(* PLC project tri_chain, Dassault Systèmes ControlBuild 2024x *)
(* stored: creationDateTime 2023-10-05T15:45:14-01:00 *)

CONFIGURATION tri_chain
  VAR_GLOBAL
    simuperiod : REAL := 50000.0;
    taskname : STRING(50) := 'tri_chain.exe';
    allowpreconditions : BOOL := true;
    allowpostconditions : BOOL := true;
    op_trichain/creation1/status_act_prod : DINT := 0;
    op_trichain/creation1/m11 : REAL := 1502.68;
    op_trichain/creation1/m12 : REAL := 0.0;
    op_trichain/creation1/m13 : REAL := -2.44921e-14;
    op_trichain/creation1/m14 : REAL := 5480.36;
    op_trichain/creation1/m21 : REAL := 0.0;
    op_trichain/creation1/m22 : REAL := 2997.32;
    op_trichain/creation1/m23 : REAL := 0.0;
    op_trichain/creation1/m24 : REAL := 27006.2;
    op_trichain/creation1/m31 : REAL := 3.68038e-13;
    op_trichain/creation1/m32 : REAL := 0.0;
    op_trichain/creation1/m33 : REAL := 100.0;
    op_trichain/creation1/m34 : REAL := 1.0;
    op_trichain/creation1/m41 : REAL := 0.0;
    op_trichain/creation1/m42 : REAL := 0.0;
    op_trichain/creation1/m43 : REAL := 0.0;
    op_trichain/creation1/m44 : REAL := 1.0;
    op_trichain/creation1/px : REAL := 5600.0;
    op_trichain/creation1/py : REAL := 27000.0;
    op_trichain/creation1/pz : REAL := 1.5;
    op_trichain/creation1/dx : REAL := 1500.0;
    op_trichain/creation1/dy : REAL := 3000.0;
    op_trichain/creation1/dz : REAL := 100.0;
    op_trichain/creation1/pulseType : BOOL := true;
    op_trichain/chain1/motor1dir/nominalSpeed : REAL := 500.0;
    op_trichain/chain1/motor1dir/nominalTime : REAL := 0.1;
    op_trichain/chain1/start_sensor/status_act_prod : DINT := 0;
    op_trichain/chain1/start_sensor/m11 : REAL := 498.214;
    op_trichain/chain1/start_sensor/m12 : REAL := 0.0;
    op_trichain/chain1/start_sensor/m13 : REAL := -2.44921e-14;
    op_trichain/chain1/start_sensor/m14 : REAL := 5223.22;
    op_trichain/chain1/start_sensor/m21 : REAL := 0.0;
    op_trichain/chain1/start_sensor/m22 : REAL := 498.214;
    op_trichain/chain1/start_sensor/m23 : REAL := 0.0;
    op_trichain/chain1/start_sensor/m24 : REAL := 26998.2;
    op_trichain/chain1/start_sensor/m31 : REAL := 1.22023e-13;
    op_trichain/chain1/start_sensor/m32 : REAL := 0.0;
    op_trichain/chain1/start_sensor/m33 : REAL := 100.0;
    op_trichain/chain1/start_sensor/m34 : REAL := 1.0;
    op_trichain/chain1/start_sensor/m41 : REAL := 0.0;
    op_trichain/chain1/start_sensor/m42 : REAL := 0.0;
    op_trichain/chain1/start_sensor/m43 : REAL := 0.0;
    op_trichain/chain1/start_sensor/m44 : REAL := 1.0;
    op_trichain/chain1/start_sensor/px : REAL := 4500.0;
    op_trichain/chain1/start_sensor/py : REAL := 27000.0;
    op_trichain/chain1/start_sensor/dx : REAL := 500.0;
    op_trichain/chain1/start_sensor/dy : REAL := 500.0;
    op_trichain/chain1/start_sensor/dz : REAL := 100.0;
    op_trichain/chain1/end_sensor/status_act_prod : DINT := 0;
    op_trichain/chain1/end_sensor/m11 : REAL := 498.214;
    op_trichain/chain1/end_sensor/m12 : REAL := 0.0;
    op_trichain/chain1/end_sensor/m13 : REAL := -2.44921e-14;
    op_trichain/chain1/end_sensor/m14 : REAL := 3334.82;
    op_trichain/chain1/end_sensor/m21 : REAL := 0.0;
    op_trichain/chain1/end_sensor/m22 : REAL := 498.214;
    op_trichain/chain1/end_sensor/m23 : REAL := 0.0;
    op_trichain/chain1/end_sensor/m24 : REAL := 19999.1;
    op_trichain/chain1/end_sensor/m31 : REAL := 1.22023e-13;
    op_trichain/chain1/end_sensor/m32 : REAL := 0.0;
    op_trichain/chain1/end_sensor/m33 : REAL := 100.0;
    op_trichain/chain1/end_sensor/m34 : REAL := 1.05;
    op_trichain/chain1/end_sensor/m41 : REAL := 0.0;
    op_trichain/chain1/end_sensor/m42 : REAL := 0.0;
    op_trichain/chain1/end_sensor/m43 : REAL := 0.0;
    op_trichain/chain1/end_sensor/m44 : REAL := 1.0;
    op_trichain/chain1/end_sensor/px : REAL := 2850.0;
    op_trichain/chain1/end_sensor/py : REAL := 20000.0;
    op_trichain/chain1/end_sensor/dx : REAL := 500.0;
    op_trichain/chain1/end_sensor/dy : REAL := 500.0;
    op_trichain/chain1/end_sensor/dz : REAL := 100.0;
    op_trichain/chain1/chain/status_act_prod : DINT := 0;
    op_trichain/chain1/chain/m11 : REAL := 4001.79;
    op_trichain/chain1/chain/m12 : REAL := 0.0;
    op_trichain/chain1/chain/m13 : REAL := -2.44921e-14;
    op_trichain/chain1/chain/m14 : REAL := 2981.25;
    op_trichain/chain1/chain/m21 : REAL := 0.0;
    op_trichain/chain1/chain/m22 : REAL := 9996.43;
    op_trichain/chain1/chain/m23 : REAL := 0.0;
    op_trichain/chain1/chain/m24 : REAL := 18102.7;
    op_trichain/chain1/chain/m31 : REAL := 9.80123e-13;
    op_trichain/chain1/chain/m32 : REAL := 0.0;
    op_trichain/chain1/chain/m33 : REAL := 100.0;
    op_trichain/chain1/chain/m34 : REAL := 1.0;
    op_trichain/chain1/chain/m41 : REAL := 0.0;
    op_trichain/chain1/chain/m42 : REAL := 0.0;
    op_trichain/chain1/chain/m43 : REAL := 0.0;
    op_trichain/chain1/chain/m44 : REAL := 1.0;
    op_trichain/chain1/chain/px : REAL := 2500.0;
    op_trichain/chain1/chain/py : REAL := 18100.0;
    op_trichain/chain1/chain/pz : REAL := 1.0;
    op_trichain/chain1/chain/dx : REAL := 4000.0;
    op_trichain/chain1/chain/dy : REAL := 10000.0;
    op_trichain/chain1/chain/dz : REAL := 100.0;
    op_trichain/chain2/motor1dir/nominalSpeed : REAL := 500.0;
    op_trichain/chain2/motor1dir/nominalTime : REAL := 0.1;
    op_trichain/chain2/start_sensor/status_act_prod : DINT := 0;
    op_trichain/chain2/start_sensor/m11 : REAL := 500.0;
    op_trichain/chain2/start_sensor/m12 : REAL := 0.0;
    op_trichain/chain2/start_sensor/m13 : REAL := 0.0;
    op_trichain/chain2/start_sensor/m14 : REAL := 8500.0;
    op_trichain/chain2/start_sensor/m21 : REAL := 0.0;
    op_trichain/chain2/start_sensor/m22 : REAL := 500.0;
    op_trichain/chain2/start_sensor/m23 : REAL := 0.0;
    op_trichain/chain2/start_sensor/m24 : REAL := 27000.0;
    op_trichain/chain2/start_sensor/m31 : REAL := 0.0;
    op_trichain/chain2/start_sensor/m32 : REAL := 0.0;
    op_trichain/chain2/start_sensor/m33 : REAL := 100.0;
    op_trichain/chain2/start_sensor/m34 : REAL := 0.0;
    op_trichain/chain2/start_sensor/m41 : REAL := 0.0;
    op_trichain/chain2/start_sensor/m42 : REAL := 0.0;
    op_trichain/chain2/start_sensor/m43 : REAL := 0.0;
    op_trichain/chain2/start_sensor/m44 : REAL := 1.0;
    op_trichain/chain2/start_sensor/px : REAL := 8500.0;
    op_trichain/chain2/start_sensor/py : REAL := 27000.0;
    op_trichain/chain2/start_sensor/dx : REAL := 500.0;
    op_trichain/chain2/start_sensor/dy : REAL := 500.0;
    op_trichain/chain2/start_sensor/dz : REAL := 100.0;
    op_trichain/chain2/end_sensor/status_act_prod : DINT := 0;
    op_trichain/chain2/end_sensor/m11 : REAL := 500.0;
    op_trichain/chain2/end_sensor/m12 : REAL := 0.0;
    op_trichain/chain2/end_sensor/m13 : REAL := 0.0;
    op_trichain/chain2/end_sensor/m14 : REAL := 6900.0;
    op_trichain/chain2/end_sensor/m21 : REAL := 0.0;
    op_trichain/chain2/end_sensor/m22 : REAL := 500.0;
    op_trichain/chain2/end_sensor/m23 : REAL := 0.0;
    op_trichain/chain2/end_sensor/m24 : REAL := 20000.0;
    op_trichain/chain2/end_sensor/m31 : REAL := 0.0;
    op_trichain/chain2/end_sensor/m32 : REAL := 0.0;
    op_trichain/chain2/end_sensor/m33 : REAL := 100.0;
    op_trichain/chain2/end_sensor/m34 : REAL := 0.0;
    op_trichain/chain2/end_sensor/m41 : REAL := 0.0;
    op_trichain/chain2/end_sensor/m42 : REAL := 0.0;
    op_trichain/chain2/end_sensor/m43 : REAL := 0.0;
    op_trichain/chain2/end_sensor/m44 : REAL := 1.0;
    op_trichain/chain2/end_sensor/px : REAL := 6900.0;
    op_trichain/chain2/end_sensor/py : REAL := 20000.0;
    op_trichain/chain2/end_sensor/dx : REAL := 500.0;
    op_trichain/chain2/end_sensor/dy : REAL := 500.0;
    op_trichain/chain2/end_sensor/dz : REAL := 100.0;
    op_trichain/chain2/chain/status_act_prod : DINT := 0;
    op_trichain/chain2/chain/m11 : REAL := 4000.0;
    op_trichain/chain2/chain/m12 : REAL := 0.0;
    op_trichain/chain2/chain/m13 : REAL := 0.0;
    op_trichain/chain2/chain/m14 : REAL := 6500.0;
    op_trichain/chain2/chain/m21 : REAL := 0.0;
    op_trichain/chain2/chain/m22 : REAL := 10000.0;
    op_trichain/chain2/chain/m23 : REAL := 0.0;
    op_trichain/chain2/chain/m24 : REAL := 18100.0;
    op_trichain/chain2/chain/m31 : REAL := 0.0;
    op_trichain/chain2/chain/m32 : REAL := 0.0;
    op_trichain/chain2/chain/m33 : REAL := 100.0;
    op_trichain/chain2/chain/m34 : REAL := 0.0;
    op_trichain/chain2/chain/m41 : REAL := 0.0;
    op_trichain/chain2/chain/m42 : REAL := 0.0;
    op_trichain/chain2/chain/m43 : REAL := 0.0;
    op_trichain/chain2/chain/m44 : REAL := 1.0;
    op_trichain/chain2/chain/px : REAL := 6500.0;
    op_trichain/chain2/chain/py : REAL := 18100.0;
    op_trichain/chain2/chain/dx : REAL := 4000.0;
    op_trichain/chain2/chain/dy : REAL := 10000.0;
    op_trichain/chain2/chain/dz : REAL := 100.0;
    op_trichain/creation2/status_act_prod : DINT := 0;
    op_trichain/creation2/m11 : REAL := 1500.0;
    op_trichain/creation2/m12 : REAL := 0.0;
    op_trichain/creation2/m13 : REAL := 0.0;
    op_trichain/creation2/m14 : REAL := 9000.0;
    op_trichain/creation2/m21 : REAL := 0.0;
    op_trichain/creation2/m22 : REAL := 3000.0;
    op_trichain/creation2/m23 : REAL := 0.0;
    op_trichain/creation2/m24 : REAL := 27000.0;
    op_trichain/creation2/m31 : REAL := 0.0;
    op_trichain/creation2/m32 : REAL := 0.0;
    op_trichain/creation2/m33 : REAL := 100.0;
    op_trichain/creation2/m34 : REAL := 0.0;
    op_trichain/creation2/m41 : REAL := 0.0;
    op_trichain/creation2/m42 : REAL := 0.0;
    op_trichain/creation2/m43 : REAL := 0.0;
    op_trichain/creation2/m44 : REAL := 1.0;
    op_trichain/creation2/px : REAL := 8990.0;
    op_trichain/creation2/py : REAL := 27000.0;
    op_trichain/creation2/pz : REAL := 1.5;
    op_trichain/creation2/dx : REAL := 1500.0;
    op_trichain/creation2/dy : REAL := 3000.0;
    op_trichain/creation2/dz : REAL := 100.0;
    op_trichain/creation2/pulseType : BOOL := true;
    op_trichain/chain3/motor1dir/nominalSpeed : REAL := 500.0;
    op_trichain/chain3/motor1dir/nominalTime : REAL := 0.1;
    op_trichain/chain3/start_sensor/status_act_prod : DINT := 0;
    op_trichain/chain3/start_sensor/m11 : REAL := 500.0;
    op_trichain/chain3/start_sensor/m12 : REAL := 0.0;
    op_trichain/chain3/start_sensor/m13 : REAL := 0.0;
    op_trichain/chain3/start_sensor/m14 : REAL := 12500.0;
    op_trichain/chain3/start_sensor/m21 : REAL := 0.0;
    op_trichain/chain3/start_sensor/m22 : REAL := 500.0;
    op_trichain/chain3/start_sensor/m23 : REAL := 0.0;
    op_trichain/chain3/start_sensor/m24 : REAL := 27000.0;
    op_trichain/chain3/start_sensor/m31 : REAL := 0.0;
    op_trichain/chain3/start_sensor/m32 : REAL := 0.0;
    op_trichain/chain3/start_sensor/m33 : REAL := 100.0;
    op_trichain/chain3/start_sensor/m34 : REAL := 0.0;
    op_trichain/chain3/start_sensor/m41 : REAL := 0.0;
    op_trichain/chain3/start_sensor/m42 : REAL := 0.0;
    op_trichain/chain3/start_sensor/m43 : REAL := 0.0;
    op_trichain/chain3/start_sensor/m44 : REAL := 1.0;
    op_trichain/chain3/start_sensor/px : REAL := 12500.0;
    op_trichain/chain3/start_sensor/py : REAL := 27000.0;
    op_trichain/chain3/start_sensor/dx : REAL := 500.0;
    op_trichain/chain3/start_sensor/dy : REAL := 500.0;
    op_trichain/chain3/start_sensor/dz : REAL := 100.0;
    op_trichain/chain3/end_sensor/status_act_prod : DINT := 0;
    op_trichain/chain3/end_sensor/m11 : REAL := 500.0;
    op_trichain/chain3/end_sensor/m12 : REAL := 0.0;
    op_trichain/chain3/end_sensor/m13 : REAL := 0.0;
    op_trichain/chain3/end_sensor/m14 : REAL := 10950.0;
    op_trichain/chain3/end_sensor/m21 : REAL := 0.0;
    op_trichain/chain3/end_sensor/m22 : REAL := 500.0;
    op_trichain/chain3/end_sensor/m23 : REAL := 0.0;
    op_trichain/chain3/end_sensor/m24 : REAL := 20000.0;
    op_trichain/chain3/end_sensor/m31 : REAL := 0.0;
    op_trichain/chain3/end_sensor/m32 : REAL := 0.0;
    op_trichain/chain3/end_sensor/m33 : REAL := 100.0;
    op_trichain/chain3/end_sensor/m34 : REAL := 0.0;
    op_trichain/chain3/end_sensor/m41 : REAL := 0.0;
    op_trichain/chain3/end_sensor/m42 : REAL := 0.0;
    op_trichain/chain3/end_sensor/m43 : REAL := 0.0;
    op_trichain/chain3/end_sensor/m44 : REAL := 1.0;
    op_trichain/chain3/end_sensor/px : REAL := 10950.0;
    op_trichain/chain3/end_sensor/py : REAL := 20000.0;
    op_trichain/chain3/chain/status_act_prod : DINT := 0;
    op_trichain/chain3/chain/m11 : REAL := 4000.0;
    op_trichain/chain3/chain/m12 : REAL := 0.0;
    op_trichain/chain3/chain/m13 : REAL := 0.0;
    op_trichain/chain3/chain/m14 : REAL := 10500.0;
    op_trichain/chain3/chain/m21 : REAL := 0.0;
    op_trichain/chain3/chain/m22 : REAL := 10000.0;
    op_trichain/chain3/chain/m23 : REAL := 0.0;
    op_trichain/chain3/chain/m24 : REAL := 18100.0;
    op_trichain/chain3/chain/m31 : REAL := 0.0;
    op_trichain/chain3/chain/m32 : REAL := 0.0;
    op_trichain/chain3/chain/m33 : REAL := 100.0;
    op_trichain/chain3/chain/m34 : REAL := 0.0;
    op_trichain/chain3/chain/m41 : REAL := 0.0;
    op_trichain/chain3/chain/m42 : REAL := 0.0;
    op_trichain/chain3/chain/m43 : REAL := 0.0;
    op_trichain/chain3/chain/m44 : REAL := 1.0;
    op_trichain/chain3/chain/px : REAL := 10500.0;
    op_trichain/chain3/chain/py : REAL := 18100.0;
    op_trichain/chain3/chain/dx : REAL := 4000.0;
    op_trichain/chain3/chain/dy : REAL := 10000.0;
    op_trichain/chain3/chain/dz : REAL := 100.0;
    op_trichain/outputChain/motor1dir/nominalSpeed : REAL := 500.0;
    op_trichain/outputChain/motor1dir/nominalTime : REAL := 0.1;
    op_trichain/outputChain/start_sensor/status_act_prod : DINT := 0;
    op_trichain/outputChain/start_sensor/m11 : REAL := 498.214;
    op_trichain/outputChain/start_sensor/m12 : REAL := 0.0;
    op_trichain/outputChain/start_sensor/m13 : REAL := 0.0;
    op_trichain/outputChain/start_sensor/m14 : REAL := 9675.0;
    op_trichain/outputChain/start_sensor/m21 : REAL := 0.0;
    op_trichain/outputChain/start_sensor/m22 : REAL := 498.214;
    op_trichain/outputChain/start_sensor/m23 : REAL := 0.0;
    op_trichain/outputChain/start_sensor/m24 : REAL := 11987.5;
    op_trichain/outputChain/start_sensor/m31 : REAL := 0.0;
    op_trichain/outputChain/start_sensor/m32 : REAL := 0.0;
    op_trichain/outputChain/start_sensor/m33 : REAL := 100.0;
    op_trichain/outputChain/start_sensor/m34 : REAL := 1.06;
    op_trichain/outputChain/start_sensor/m41 : REAL := 0.0;
    op_trichain/outputChain/start_sensor/m42 : REAL := 0.0;
    op_trichain/outputChain/start_sensor/m43 : REAL := 0.0;
    op_trichain/outputChain/start_sensor/m44 : REAL := 1.0;
    op_trichain/outputChain/start_sensor/dx : REAL := 500.0;
    op_trichain/outputChain/start_sensor/dy : REAL := 500.0;
    op_trichain/outputChain/start_sensor/dz : REAL := 100.0;
    op_trichain/outputChain/end_sensor/status_act_prod : DINT := 0;
    op_trichain/outputChain/end_sensor/m11 : REAL := 500.0;
    op_trichain/outputChain/end_sensor/m12 : REAL := 0.0;
    op_trichain/outputChain/end_sensor/m13 : REAL := 0.0;
    op_trichain/outputChain/end_sensor/m14 : REAL := 7450.0;
    op_trichain/outputChain/end_sensor/m21 : REAL := 0.0;
    op_trichain/outputChain/end_sensor/m22 : REAL := 500.0;
    op_trichain/outputChain/end_sensor/m23 : REAL := 0.0;
    op_trichain/outputChain/end_sensor/m24 : REAL := 4800.0;
    op_trichain/outputChain/end_sensor/m31 : REAL := 0.0;
    op_trichain/outputChain/end_sensor/m32 : REAL := 0.0;
    op_trichain/outputChain/end_sensor/m33 : REAL := 100.0;
    op_trichain/outputChain/end_sensor/m34 : REAL := 1.0;
    op_trichain/outputChain/end_sensor/m41 : REAL := 0.0;
    op_trichain/outputChain/end_sensor/m42 : REAL := 0.0;
    op_trichain/outputChain/end_sensor/m43 : REAL := 0.0;
    op_trichain/outputChain/end_sensor/m44 : REAL := 1.0;
    op_trichain/outputChain/end_sensor/px : REAL := 7450.0;
    op_trichain/outputChain/end_sensor/py : REAL := 4800.0;
    op_trichain/outputChain/end_sensor/dx : REAL := 500.0;
    op_trichain/outputChain/end_sensor/dy : REAL := 500.0;
    op_trichain/outputChain/end_sensor/dz : REAL := 100.0;
    op_trichain/outputChain/chain/status_act_prod : DINT := 0;
    op_trichain/outputChain/chain/m11 : REAL := 4001.79;
    op_trichain/outputChain/chain/m12 : REAL := 0.0;
    op_trichain/outputChain/chain/m13 : REAL := 0.0;
    op_trichain/outputChain/chain/m14 : REAL := 7003.57;
    op_trichain/outputChain/chain/m21 : REAL := 0.0;
    op_trichain/outputChain/chain/m22 : REAL := 9996.43;
    op_trichain/outputChain/chain/m23 : REAL := 0.0;
    op_trichain/outputChain/chain/m24 : REAL := 2352.06;
    op_trichain/outputChain/chain/m31 : REAL := 0.0;
    op_trichain/outputChain/chain/m32 : REAL := 0.0;
    op_trichain/outputChain/chain/m33 : REAL := 100.0;
    op_trichain/outputChain/chain/m34 : REAL := 1.06;
    op_trichain/outputChain/chain/m41 : REAL := 0.0;
    op_trichain/outputChain/chain/m42 : REAL := 0.0;
    op_trichain/outputChain/chain/m43 : REAL := 0.0;
    op_trichain/outputChain/chain/m44 : REAL := 1.0;
    op_trichain/outputChain/chain/px : REAL := 7100.0;
    op_trichain/outputChain/chain/py : REAL := 3000.0;
    op_trichain/outputChain/chain/dx : REAL := 4000.0;
    op_trichain/outputChain/chain/dy : REAL := 10000.0;
    op_trichain/outputChain/chain/dz : REAL := 100.0;
    op_trichain/shuttle/motor2dir/nominalSpeed : REAL := 500.0;
    op_trichain/shuttle/motor2dir/nominalTime : REAL := 0.1;
    op_trichain/shuttle/chainMotor/nominalSpeed : REAL := 500.0;
    op_trichain/shuttle/chainMotor/nominalTime : REAL := 0.1;
    op_trichain/shuttle/axle/initTranslat : REAL := 5100.0;
    op_trichain/shuttle/axle/maxTranslat : REAL := 30000.0;
    op_trichain/shuttle/shuttle/status_act_prod : DINT := 0;
    op_trichain/shuttle/shuttle/m11 : REAL := 2997.32;
    op_trichain/shuttle/shuttle/m12 : REAL := 0.0;
    op_trichain/shuttle/shuttle/m13 : REAL := -2.44921e-14;
    op_trichain/shuttle/shuttle/m14 : REAL := 5231.25;
    op_trichain/shuttle/shuttle/m21 : REAL := 0.0;
    op_trichain/shuttle/shuttle/m22 : REAL := 7497.32;
    op_trichain/shuttle/shuttle/m23 : REAL := 0.0;
    op_trichain/shuttle/shuttle/m24 : REAL := 11601.8;
    op_trichain/shuttle/shuttle/m31 : REAL := 7.34108e-13;
    op_trichain/shuttle/shuttle/m32 : REAL := 0.0;
    op_trichain/shuttle/shuttle/m33 : REAL := 100.0;
    op_trichain/shuttle/shuttle/m34 : REAL := 1.05;
    op_trichain/shuttle/shuttle/m41 : REAL := 0.0;
    op_trichain/shuttle/shuttle/m42 : REAL := 0.0;
    op_trichain/shuttle/shuttle/m43 : REAL := 0.0;
    op_trichain/shuttle/shuttle/m44 : REAL := 1.0;
    op_trichain/shuttle/shuttle/px : REAL := 5250.0;
    op_trichain/shuttle/shuttle/py : REAL := 11600.0;
    op_trichain/shuttle/shuttle/pz : REAL := 1.05;
    op_trichain/shuttle/shuttle/dx : REAL := 3000.0;
    op_trichain/shuttle/shuttle/dy : REAL := 7500.0;
    op_trichain/shuttle/shuttle/dz : REAL := 100.0;
    op_trichain/shuttle/pos1Sensor/status_act_prod : DINT := 0;
    op_trichain/shuttle/pos1Sensor/m11 : REAL := 498.214;
    op_trichain/shuttle/pos1Sensor/m12 : REAL := 0.0;
    op_trichain/shuttle/pos1Sensor/m13 : REAL := 0.0;
    op_trichain/shuttle/pos1Sensor/m14 : REAL := 3479.47;
    op_trichain/shuttle/pos1Sensor/m21 : REAL := 0.0;
    op_trichain/shuttle/pos1Sensor/m22 : REAL := 498.214;
    op_trichain/shuttle/pos1Sensor/m23 : REAL := 0.0;
    op_trichain/shuttle/pos1Sensor/m24 : REAL := 17998.2;
    op_trichain/shuttle/pos1Sensor/m31 : REAL := 0.0;
    op_trichain/shuttle/pos1Sensor/m32 : REAL := 0.0;
    op_trichain/shuttle/pos1Sensor/m33 : REAL := 100.0;
    op_trichain/shuttle/pos1Sensor/m34 : REAL := 1.05;
    op_trichain/shuttle/pos1Sensor/m41 : REAL := 0.0;
    op_trichain/shuttle/pos1Sensor/m42 : REAL := 0.0;
    op_trichain/shuttle/pos1Sensor/m43 : REAL := 0.0;
    op_trichain/shuttle/pos1Sensor/m44 : REAL := 1.0;
    op_trichain/shuttle/pos1Sensor/threshold : REAL := 900.0;
    op_trichain/shuttle/pos1Sensor/range : REAL := 900.0;
    op_trichain/shuttle/pos2Sensor/status_act_prod : DINT := 0;
    op_trichain/shuttle/pos2Sensor/m11 : REAL := 500.0;
    op_trichain/shuttle/pos2Sensor/m12 : REAL := 0.0;
    op_trichain/shuttle/pos2Sensor/m13 : REAL := 0.0;
    op_trichain/shuttle/pos2Sensor/m14 : REAL := 7000.0;
    op_trichain/shuttle/pos2Sensor/m21 : REAL := 0.0;
    op_trichain/shuttle/pos2Sensor/m22 : REAL := 500.0;
    op_trichain/shuttle/pos2Sensor/m23 : REAL := 0.0;
    op_trichain/shuttle/pos2Sensor/m24 : REAL := 18000.0;
    op_trichain/shuttle/pos2Sensor/m31 : REAL := 0.0;
    op_trichain/shuttle/pos2Sensor/m32 : REAL := 0.0;
    op_trichain/shuttle/pos2Sensor/m33 : REAL := 100.0;
    op_trichain/shuttle/pos2Sensor/m34 : REAL := 1.06;
    op_trichain/shuttle/pos2Sensor/m41 : REAL := 0.0;
    op_trichain/shuttle/pos2Sensor/m42 : REAL := 0.0;
    op_trichain/shuttle/pos2Sensor/m43 : REAL := 0.0;
    op_trichain/shuttle/pos2Sensor/m44 : REAL := 1.0;
    op_trichain/shuttle/pos2Sensor/threshold : REAL := 4500.0;
    op_trichain/shuttle/pos2Sensor/range : REAL := 900.0;
    op_trichain/shuttle/pos3Sensor/status_act_prod : DINT := 0;
    op_trichain/shuttle/pos3Sensor/m11 : REAL := 500.0;
    op_trichain/shuttle/pos3Sensor/m12 : REAL := 0.0;
    op_trichain/shuttle/pos3Sensor/m13 : REAL := 0.0;
    op_trichain/shuttle/pos3Sensor/m14 : REAL := 11400.0;
    op_trichain/shuttle/pos3Sensor/m21 : REAL := 0.0;
    op_trichain/shuttle/pos3Sensor/m22 : REAL := 500.0;
    op_trichain/shuttle/pos3Sensor/m23 : REAL := 0.0;
    op_trichain/shuttle/pos3Sensor/m24 : REAL := 18000.0;
    op_trichain/shuttle/pos3Sensor/m31 : REAL := 0.0;
    op_trichain/shuttle/pos3Sensor/m32 : REAL := 0.0;
    op_trichain/shuttle/pos3Sensor/m33 : REAL := 100.0;
    op_trichain/shuttle/pos3Sensor/m34 : REAL := 0.0;
    op_trichain/shuttle/pos3Sensor/m41 : REAL := 0.0;
    op_trichain/shuttle/pos3Sensor/m42 : REAL := 0.0;
    op_trichain/shuttle/pos3Sensor/m43 : REAL := 0.0;
    op_trichain/shuttle/pos3Sensor/m44 : REAL := 1.0;
    op_trichain/shuttle/pos3Sensor/threshold : REAL := 9200.0;
    op_trichain/shuttle/pos3Sensor/range : REAL := 900.0;
    op_trichain/shuttle/endSensor/status_act_prod : DINT := 0;
    op_trichain/shuttle/endSensor/m11 : REAL := 337.5;
    op_trichain/shuttle/endSensor/m12 : REAL := 0.0;
    op_trichain/shuttle/endSensor/m13 : REAL := 0.0;
    op_trichain/shuttle/endSensor/m14 : REAL := 5464.29;
    op_trichain/shuttle/endSensor/m21 : REAL := 0.0;
    op_trichain/shuttle/endSensor/m22 : REAL := 369.643;
    op_trichain/shuttle/endSensor/m23 : REAL := 0.0;
    op_trichain/shuttle/endSensor/m24 : REAL := 13032.1;
    op_trichain/shuttle/endSensor/m31 : REAL := 0.0;
    op_trichain/shuttle/endSensor/m32 : REAL := 0.0;
    op_trichain/shuttle/endSensor/m33 : REAL := 100.0;
    op_trichain/shuttle/endSensor/m34 : REAL := 1.0;
    op_trichain/shuttle/endSensor/m41 : REAL := 0.0;
    op_trichain/shuttle/endSensor/m42 : REAL := 0.0;
    op_trichain/shuttle/endSensor/m43 : REAL := 0.0;
    op_trichain/shuttle/endSensor/m44 : REAL := 1.0;
    op_trichain/shuttle/endSensor/py : REAL := 14500.0;
    op_trichain/shuttle/endSensor/dx : REAL := 500.0;
    op_trichain/shuttle/endSensor/dy : REAL := 500.0;
    op_trichain/shuttle/endSensor/dz : REAL := 100.0;
    op_trichain/shuttle/endSensor/initialPosition : REAL := 1000.0;
    op_trichain/creation3/status_act_prod : DINT := 0;
    op_trichain/creation3/m11 : REAL := 1500.0;
    op_trichain/creation3/m12 : REAL := 0.0;
    op_trichain/creation3/m13 : REAL := 0.0;
    op_trichain/creation3/m14 : REAL := 13000.0;
    op_trichain/creation3/m21 : REAL := 0.0;
    op_trichain/creation3/m22 : REAL := 3000.0;
    op_trichain/creation3/m23 : REAL := 0.0;
    op_trichain/creation3/m24 : REAL := 27000.0;
    op_trichain/creation3/m31 : REAL := 0.0;
    op_trichain/creation3/m32 : REAL := 0.0;
    op_trichain/creation3/m33 : REAL := 100.0;
    op_trichain/creation3/m34 : REAL := 0.0;
    op_trichain/creation3/m41 : REAL := 0.0;
    op_trichain/creation3/m42 : REAL := 0.0;
    op_trichain/creation3/m43 : REAL := 0.0;
    op_trichain/creation3/m44 : REAL := 1.0;
    op_trichain/creation3/px : REAL := 12990.0;
    op_trichain/creation3/py : REAL := 27000.0;
    op_trichain/creation3/pz : REAL := 1.5;
    op_trichain/creation3/dx : REAL := 1500.0;
    op_trichain/creation3/dy : REAL := 3000.0;
    op_trichain/creation3/dz : REAL := 100.0;
    op_trichain/creation3/pulseType : BOOL := true;
    op_trichain/trash/status_act_prod : DINT := 0;
    op_trichain/trash/m11 : REAL := 1197.32;
    op_trichain/trash/m12 : REAL := 0.0;
    op_trichain/trash/m13 : REAL := -2.44921e-14;
    op_trichain/trash/m14 : REAL := 7103.57;
    op_trichain/trash/m21 : REAL := 0.0;
    op_trichain/trash/m22 : REAL := 2499.11;
    op_trichain/trash/m23 : REAL := 0.0;
    op_trichain/trash/m24 : REAL := 841.954;
    op_trichain/trash/m31 : REAL := 2.9325e-13;
    op_trichain/trash/m32 : REAL := 0.0;
    op_trichain/trash/m33 : REAL := 100.0;
    op_trichain/trash/m34 : REAL := 1.0;
    op_trichain/trash/m41 : REAL := 0.0;
    op_trichain/trash/m42 : REAL := 0.0;
    op_trichain/trash/m43 : REAL := 0.0;
    op_trichain/trash/m44 : REAL := 1.0;
    op_trichain/trash/px : REAL := 7100.0;
    op_trichain/trash/py : REAL := 1400.0;
    op_trichain/trash/dx : REAL := 1200.0;
    op_trichain/trash/dy : REAL := 2500.0;
    op_trichain/trash/dz : REAL := 100.0;
  END_VAR
END_CONFIGURATION
